FUNCTION_BLOCK GetBlueprintVisitor
VAR
	response : I_Serializer;
END_VAR

METHOD FB_init : BOOL
VAR_INPUT
	bInitRetains : BOOL; // if TRUE, the retain variables are initialized (warm start / cold start)
	bInCopyCode : BOOL;  // if TRUE, the instance afterwards gets moved into the copy code (online change)
	Serializer : I_Serializer;
END_VAR
This^.response := Serializer;
END_METHOD

END_FUNCTION_BLOCK

(* stored: Version 1.1.0.1, ProductVersion 3.1.4024.12
   POU GetBlueprintVisitor: Id {aebd2441-509d-0d3c-0e27-d150be94dd61}, SpecialFunc None
   Folder Constructor: Id {4cbdd883-0847-0002-0a09-8fc08ea563bb}
   Folder Private: Id {6b78b35a-b566-09b1-3105-31d9b49f4ce8}
   Method FB_init: Id {0307417a-cb8f-0fb2-3c9e-ef3535e28d87} *)
